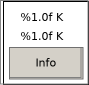
VISUALIZATION VISU_TEMP_POMP_CRYO_SOLO  // 89x85
VAR_IN_OUT
	m_Input_CRYO: BLOCK_RS232_ONBOARD_V4;
	m_Input_PRG_POMPAGE: BLOCK_PRG_POMPAGE;
END_VAR
VAR_INPUT
	m_Input_NumFrame_Manu:	USINT;		(*numéro de frame à afficher dans le synoptique MANUEL*)
	m_Input_INDEX_CRYO : INT;
END_VAR
    RoundedRectangle (3,1 86x84)
    Rectangle (7,8 70x19), "%1.0f K", text variable: PRG_POMPAGE.COM_CRYOS.STATE_Temperature[0]
    Rectangle (7,27 70x19), "%1.0f K", text variable: PRG_POMPAGE.COM_CRYOS.STATE_Temperature[1]
    Button (9,47 74x32), "Info"
        OnMouseClick: change screen: SYN_MANUEL
        OnMouseClick: execute { .VISU_INDEX_MANU := m_Input_NumFrame_Manu; }
END_VISUALIZATION

(* stored: Version 1.1.0.1, ProductVersion 3.1.4026.18
   Visu VISU_TEMP_POMP_CRYO_SOLO: Id {8c2aeafd-cbff-41b0-b83c-8e6a141d4fd7} *)
